(* LS Electric XG5000 project: Desummer *)
(* PLC LSPLC *)
(* module base 0 slot 0: FEnet:XGL-EFMT(B) (Fast Ethernet 통신 모듈, 전기 Master) *)
(* module base 0 slot 1: 입력 모듈:XGI-A21A/C (AC 220V 입력, 8점(8점/COM) / 8점(1점/COM)) *)
(* module base 0 slot 2: 출력 모듈:XGQ-RY1A (릴레이 출력, 8점 (2A용, 단독 COM.)) *)

FUNCTION_BLOCK 보온로자동제어
VAR_INPUT
    보온로온도 : WORD;
END_VAR
VAR_OUTPUT
    valve : BOOL;
    화로1_On : BOOL;
    화로2_On : BOOL;
    화로3_On : BOOL;
END_VAR
VAR
    after2s : TON;
    check : BOOL;
    for3s : TON;
    for3s_1 : TON;
    화로_제어온도_1 : WORD := 700;
    화로_제어온도_2 : WORD := 685;
    화로_제어온도_3 : WORD := 670;
END_VAR

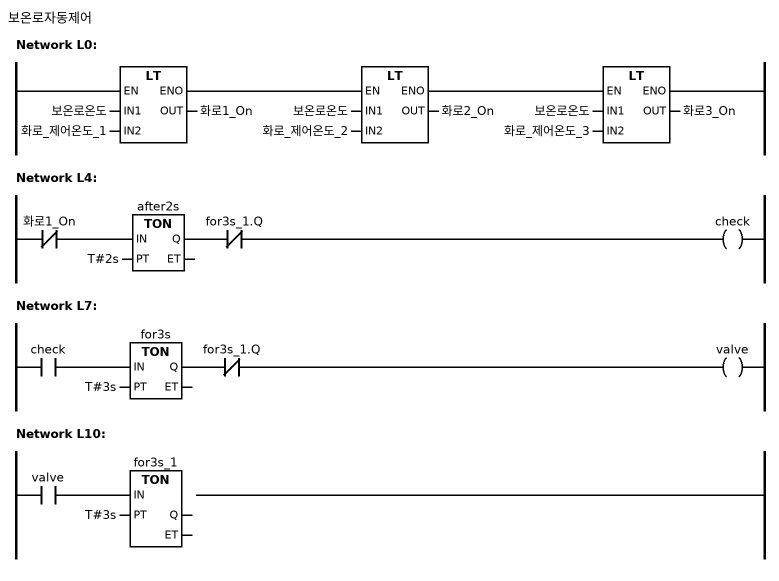
(* Rung L0 *)
화로1_On := 보온로온도 < 화로_제어온도_1;
화로2_On := 보온로온도 < 화로_제어온도_2;
화로3_On := 보온로온도 < 화로_제어온도_3;
(* Rung L4 *)
after2s(IN := NOT 화로1_On, PT := T#2s);
check := after2s.Q AND NOT for3s_1.Q;
(* Rung L7 *)
for3s(IN := check, PT := T#3s);
valve := for3s.Q AND NOT for3s_1.Q;
(* Rung L10 *)
for3s_1(IN := valve, PT := T#3s);
END_FUNCTION_BLOCK

FUNCTION_BLOCK 보온로수동제어
VAR_INPUT
    on_hot : BOOL;
    off_hot : BOOL;
    valve_input : BOOL;
    안전모드ONOFF : BOOL;
    보온로온도 : WORD;
END_VAR
VAR_OUTPUT
    hot1 : BOOL;
    hot2 : BOOL;
    hot3 : BOOL;
    valve_output : BOOL;
END_VAR
VAR
    all_off : BOOL;
    for3s : TP;
    off1 : BOOL;
    off2 : BOOL;
    off3 : BOOL;
    안전모드ON : BOOL;
END_VAR
VAR
    _e1 : R_TRIG;
    _e2 : R_TRIG;
    _e3 : R_TRIG;
    _e4 : R_TRIG;
    _e5 : R_TRIG;
    _e6 : R_TRIG;
END_VAR

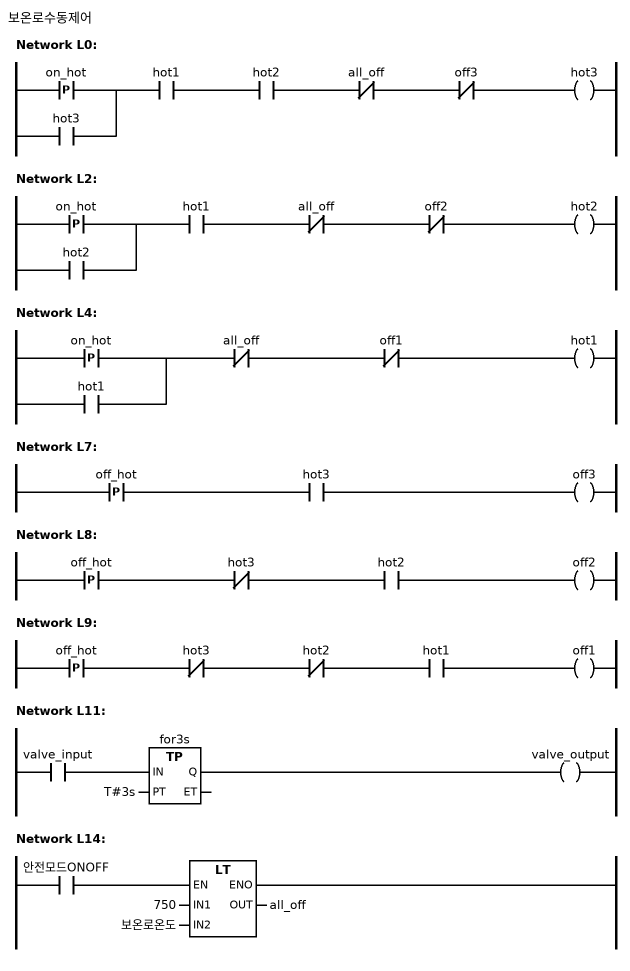
(* Rung L0 *)
_e1(CLK := on_hot);
hot3 := (_e1.Q OR hot3) AND hot1 AND hot2 AND NOT all_off AND NOT off3;
(* Rung L2 *)
_e2(CLK := on_hot);
hot2 := (_e2.Q OR hot2) AND hot1 AND NOT all_off AND NOT off2;
(* Rung L4 *)
_e3(CLK := on_hot);
hot1 := (_e3.Q OR hot1) AND NOT all_off AND NOT off1;
(* Rung L7 *)
_e4(CLK := off_hot);
off3 := _e4.Q AND hot3;
(* Rung L8 *)
_e5(CLK := off_hot);
off2 := _e5.Q AND NOT hot3 AND hot2;
(* Rung L9 *)
_e6(CLK := off_hot);
off1 := _e6.Q AND NOT hot3 AND NOT hot2 AND hot1;
(* Rung L11 *)
for3s(IN := valve_input, PT := T#3s);
valve_output := for3s.Q;
(* Rung L14 *)
IF 안전모드ONOFF THEN all_off := 750 < 보온로온도; END_IF;
END_FUNCTION_BLOCK

PROGRAM Desummer (* task: 스캔 프로그램 *)
VAR
    A밸브 AT %MX6 : BOOL;
    A보온로수동제어 : 보온로수동제어;
    A보온로온도 AT %MW200 : WORD := 701;
    A보온로자동제어 : 보온로자동제어;
    A비정상신호 AT %MX1 : BOOL;
    A수동밸브 AT %MX27 : BOOL;
    A안전모드 AT %MX30 : BOOL;
    A안전신호 AT %MX33 : BOOL;
    A자동수동설정 AT %MX9 : BOOL;
    A정상신호 AT %MX0 : BOOL;
    A화로1 AT %MX12 : BOOL;
    A화로2 AT %MX13 : BOOL;
    A화로3 AT %MX14 : BOOL;
    A화로OFF AT %MX24 : BOOL;
    A화로ON AT %MX21 : BOOL;
    B밸브 AT %MX7 : BOOL;
    B보온로수동제어 : 보온로수동제어;
    B보온로온도 AT %MW201 : WORD := 650;
    B보온로자동제어 : 보온로자동제어;
    B비정상신호 AT %MX3 : BOOL;
    B수동밸브 AT %MX28 : BOOL;
    B안전모드 AT %MX31 : BOOL;
    B안전신호 AT %MX34 : BOOL;
    B자동수동설정 AT %MX10 : BOOL;
    B정상신호 AT %MX2 : BOOL;
    B화로1 AT %MX15 : BOOL;
    B화로2 AT %MX16 : BOOL;
    B화로3 AT %MX17 : BOOL;
    B화로OFF AT %MX25 : BOOL;
    B화로ON AT %MX22 : BOOL;
    C밸브 AT %MX8 : BOOL;
    C보온로수동제어 : 보온로수동제어;
    C보온로온도 AT %MW202 : WORD := 710;
    C보온로자동제어 : 보온로자동제어;
    C비정상신호 AT %MX5 : BOOL;
    C수동밸브 AT %MX29 : BOOL;
    C안전모드 AT %MX32 : BOOL;
    C안전신호 AT %MX35 : BOOL;
    C자동수동설정 AT %MX11 : BOOL;
    C정상신호 AT %MX4 : BOOL;
    C화로1 AT %MX18 : BOOL;
    C화로2 AT %MX19 : BOOL;
    C화로3 AT %MX20 : BOOL;
    C화로OFF AT %MX26 : BOOL;
    C화로ON AT %MX23 : BOOL;
    _0번출력포트 AT %QX0.2.0 : BOOL;
    _1번출력포트 AT %QX0.2.1 : BOOL;
    _2번출력포트 AT %QX0.2.2 : BOOL;
END_VAR

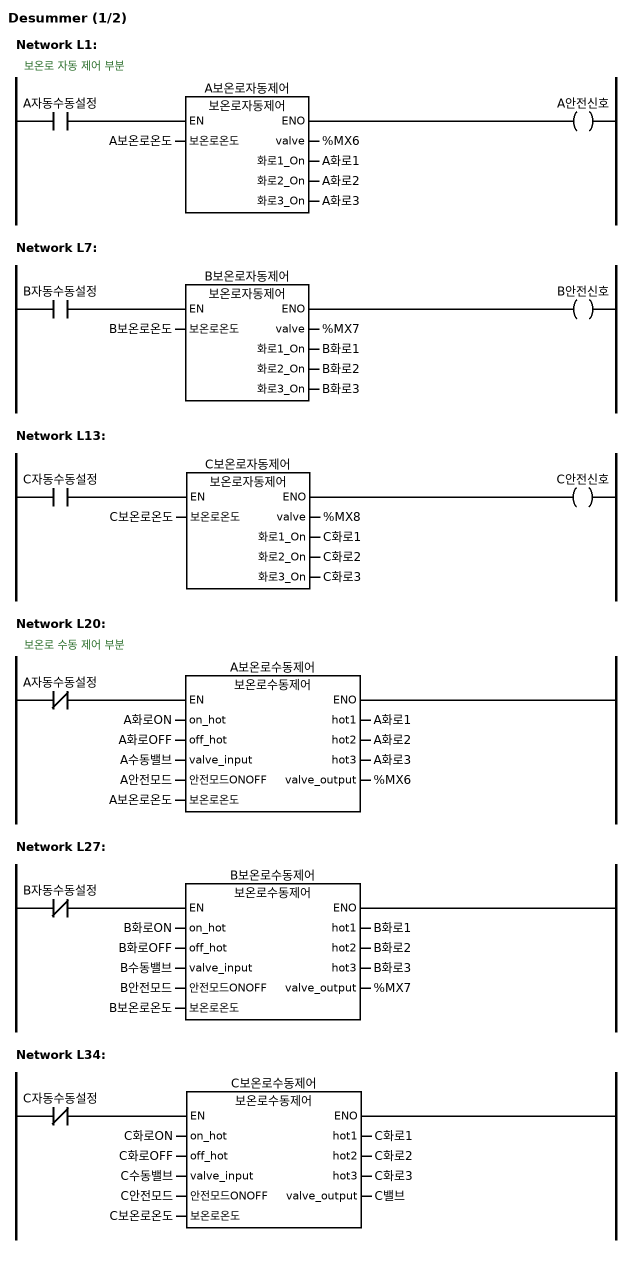
(* 보온로 자동 제어 부분 *)
(* Rung L1 *)
IF A자동수동설정 THEN
    A보온로자동제어(보온로온도 := A보온로온도, valve => %MX6, 화로1_On => A화로1, 화로2_On => A화로2, 화로3_On => A화로3);
END_IF;
A안전신호 := A자동수동설정;
(* Rung L7 *)
IF B자동수동설정 THEN
    B보온로자동제어(보온로온도 := B보온로온도, valve => %MX7, 화로1_On => B화로1, 화로2_On => B화로2, 화로3_On => B화로3);
END_IF;
B안전신호 := B자동수동설정;
(* Rung L13 *)
IF C자동수동설정 THEN
    C보온로자동제어(보온로온도 := C보온로온도, valve => %MX8, 화로1_On => C화로1, 화로2_On => C화로2, 화로3_On => C화로3);
END_IF;
C안전신호 := C자동수동설정;
(* 보온로 수동 제어 부분 *)
(* Rung L20 *)
IF NOT A자동수동설정 THEN
    A보온로수동제어(on_hot := A화로ON, off_hot := A화로OFF, valve_input := A수동밸브, 안전모드ONOFF := A안전모드, 보온로온도 := A보온로온도, hot1 => A화로1, hot2 => A화로2, hot3 => A화로3, valve_output => %MX6);
END_IF;
(* Rung L27 *)
IF NOT B자동수동설정 THEN
    B보온로수동제어(on_hot := B화로ON, off_hot := B화로OFF, valve_input := B수동밸브, 안전모드ONOFF := B안전모드, 보온로온도 := B보온로온도, hot1 => B화로1, hot2 => B화로2, hot3 => B화로3, valve_output => %MX7);
END_IF;
(* Rung L34 *)
IF NOT C자동수동설정 THEN
    C보온로수동제어(on_hot := C화로ON, off_hot := C화로OFF, valve_input := C수동밸브, 안전모드ONOFF := C안전모드, 보온로온도 := C보온로온도, hot1 => C화로1, hot2 => C화로2, hot3 => C화로3, valve_output => C밸브);
END_IF;

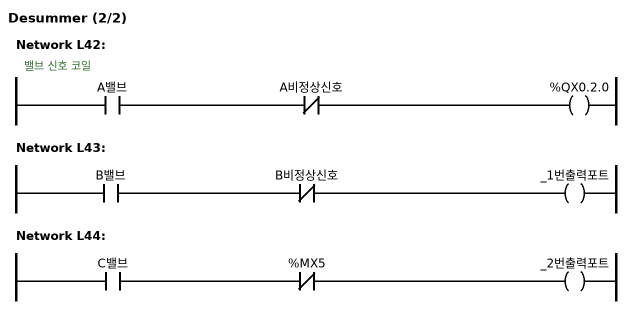
(* 밸브 신호 코일 *)
(* Rung L42 *)
%QX0.2.0 := A밸브 AND NOT A비정상신호;
(* Rung L43 *)
_1번출력포트 := B밸브 AND NOT B비정상신호;
(* Rung L44 *)
_2번출력포트 := C밸브 AND NOT %MX5;
END_PROGRAM